(*

.. <legal notes>

legal notes
=================
| SPDX-FileCopyrightText: © 2025 Oleksandr Tiutyk <trofimich@gmail.com>
| SPDX-License-Identifier: LGPL-3.0-only
| For details check: LGPL-3.0-only_

.. _LGPL-3.0-only: https://www.gnu.org/licenses/lgpl-3.0.en.html

.. </legal notes>

*)

INTERFACE IArgumentNullException EXTENDS IGeneralException

END_INTERFACE

(* stored: Version 1.1.0.1
   Itf IArgumentNullException: Id {178844c7-5cfd-43eb-805a-0df047e1434a} *)
